FUNCTION_BLOCK FB_MockGeometryWriter IMPLEMENTS I_GeometryWriter
VAR_OUTPUT
    ClearCount                     : INT;
    EnableTangentialFollowingCount : INT;
    AddStartPointCount             : INT;
    AddLineCount                   : INT;
    AddArcCount                    : INT;
    EndTableCount                  : INT;
    
    // Ostatnie parametry ze StartPoint (do weryfikacji)
    LastStartX : LREAL;
    LastStartY : LREAL;
END_VAR

METHOD AddArc : BOOL
VAR_INPUT
    TargetX    : LREAL;
    TargetY    : LREAL;
    CenterX    : LREAL;
    CenterY    : LREAL;
    Velo       : LREAL;
    Clockwise  : BOOL;
END_VAR
AddArcCount := AddArcCount + 1;
AddArc := TRUE;
END_METHOD

METHOD AddLine : BOOL
VAR_INPUT
    TargetX : LREAL;
    TargetY : LREAL;
    Velo    : LREAL;
END_VAR
AddLineCount := AddLineCount + 1;
AddLine := TRUE;
END_METHOD

METHOD AddStartPoint : BOOL
VAR_INPUT
    TargetX : LREAL;
    TargetY : LREAL;
END_VAR
AddStartPointCount := AddStartPointCount + 1;
LastStartX := TargetX;
LastStartY := TargetY;
AddStartPoint := TRUE;
END_METHOD

METHOD Clear : BOOL
VAR_INPUT
END_VAR
ClearCount := ClearCount + 1;
Clear := TRUE;
END_METHOD

METHOD EnableTangentialFollowing : BOOL
VAR_INPUT
END_VAR
EnableTangentialFollowingCount := EnableTangentialFollowingCount + 1;
EnableTangentialFollowing := TRUE;
END_METHOD

METHOD EndTable : BOOL
VAR_INPUT
END_VAR
EndTableCount := EndTableCount + 1;
EndTable := TRUE;
END_METHOD

METHOD ResetCounters
ClearCount := 0;
EnableTangentialFollowingCount := 0;
AddStartPointCount := 0;
AddLineCount := 0;
AddArcCount := 0;
EndTableCount := 0;
LastStartX := 0.0;
LastStartY := 0.0;
END_METHOD

END_FUNCTION_BLOCK

(* stored: Version 1.1.0.1, ProductVersion 3.1.4024.15
   POU FB_MockGeometryWriter: Id {a1b2c3d4-e5f6-4789-9999-10c4930e0000}, SpecialFunc None
   Method AddArc: Id {a1b2c3d4-e5f6-4789-9999-10c4930e0001}
   Method AddLine: Id {a1b2c3d4-e5f6-4789-9999-10c4930e0002}
   Method AddStartPoint: Id {a1b2c3d4-e5f6-4789-9999-10c4930e0003}
   Method Clear: Id {a1b2c3d4-e5f6-4789-9999-10c4930e0004}
   Method EnableTangentialFollowing: Id {a1b2c3d4-e5f6-4789-9999-10c4930e0005}
   Method EndTable: Id {a1b2c3d4-e5f6-4789-9999-10c4930e0006}
   Method ResetCounters: Id {a1b2c3d4-e5f6-4789-9999-10c4930e0007} *)
